// Brief: Master Arm Error Hold
FUNCTION_BLOCK PUBLIC FB_StateCtrlDisable EXTENDS FB_MasterArmCtrlBase
VAR_INPUT
END_VAR
VAR_OUTPUT
END_VAR
VAR
END_VAR

// override this function in each exact controller
METHOD PROTECTED calcCmdJntPos : BOOL

VAR_IN_OUT CONSTANT
	i_slaveIdx :INT;
	i_shoulderPose :ST_Frame;
	i_masterArm :FB_MasterArm;
	i_slaveStatus :ST_SlaveStatus;
END_VAR
var 
	i,j : INT;

	
END_VAR
m_cmdJntPos:= i_masterArm.curJntPos;
m_cmdJntVel := g_zeroVec7d;
END_METHOD

METHOD PUBLIC init : BOOL
VAR_IN_OUT CONSTANT
	i_masterArm	:FB_MasterArm;
END_VAR
VAR_IN_OUT 
	r_masterArmCtrlCmd :ST_ArmCtrlCmds;
END_VAR

VAR
	i:INT;
END_VAR
SUPER^.Init(i_masterArm,r_masterArmCtrlCmd);
m_jntOPMode:=g_allPosMode;

// disable all joints
m_jntEnableFlag :=g_zeroVec7i;
END_METHOD

END_FUNCTION_BLOCK

(* stored: Version 1.1.0.1, ProductVersion 3.1.4024.12
   POU FB_StateCtrlDisable: Id {cdb57e54-fa38-4cad-b467-29f4110c1ee2}, SpecialFunc None
   Method calcCmdJntPos: Id {89de411a-bd80-47a9-a64c-96ec6b6393ef}
   Method init: Id {7ec4f7df-df49-4afd-a16c-f71bb7ca37e5} *)
